// TIA Portal V20 export
FUNCTION "FC_AnalogInputAction" : Void   // FC1302, SCL
{ S7_Optimized_Access := 'TRUE' }
// stored: AutoNumber false, SetENOAutomatically false
   VAR_INPUT
      iReset : Bool;
   END_VAR
   VAR_OUTPUT
      oBadPartOnFixture : Bool;
      oID_MeasureBad : Int;
   END_VAR
   VAR_TEMP
      tIndex : Int;
      tResultByte0 : Int;
      tResultByte2 : Int;
      tResultByte3 : Int;
      tInitValue : LWord;
   END_VAR
BEGIN
   REGION Description header 
       //==================================================================================
       // POSALUX Swiss SA / (C) Copyright 2025
       //----------------------------------------------------------------------------------
       // Title: FC_PLC-ISO-IHM
       // Comment/Function: Manage analog variables
       //                   - BadPartOnFixture:  Set to 1 if any BadPartOnFixture bit in DB_Analog_Input_Setting = 1  
       //                                        Set to 0 if all BadPartOnFixture bits in DB_Analog_Input_Setting = 0  
       // Author: Fabien Waldt
       // Engineering: TIA Portal v17
       //----------------------------------------------------------------------------------
       // Change log table:
       // Version  | Date     | Expert in charge | Changes applied
       // ---------|----------|------------------|------------------------------------
       // 00.00.01 | 20250312 | WFA              | First released version
       // 00.00.02 | 20250807 | WFA              | Removal of the StopMachine feature
       // ==================================================================================
   END_REGION

   REGION Reset Values
       IF #iReset THEN
           #tInitValue := 0;
           FOR #tIndex := 0 TO 74 DO
               POKE(area := 16#84,
                    dbNumber := 1304,
                    byteOffset := #tIndex,
                    value := #tInitValue);
           END_FOR;
       END_IF;
   END_REGION

   REGION Bad Part On Fixture
       FOR #tIndex := 0 TO 74 BY 4 DO
           #tResultByte0 := PEEK(area := 16#84, dbNumber := 1304, byteOffset := #tIndex);
           #tResultByte2 := PEEK(area := 16#84, dbNumber := 1304, byteOffset := #tIndex + 2);
           #tResultByte3 := PEEK(area := 16#84, dbNumber := 1304, byteOffset := #tIndex + 3);
           #oBadPartOnFixture := FALSE;
           IF #tResultByte0.%X0 THEN
               #oBadPartOnFixture := TRUE;
               #oID_MeasureBad := ABS(SHL(IN := #tResultByte2, N := 8) OR #tResultByte3);
               EXIT;
           END_IF;
       END_FOR;
   END_REGION
END_FUNCTION
